PROGRAM MAIN
VAR
fbProfiler: Profiler;
stProfilerResult:PROFILERSTRUCT;
nAnsOfFactorial:ULINT;
END_VAR

fbProfiler(start:=TRUE,reset:=FALSE);
	Factorial(nAnsOfFactorial);	
fbProfiler(start:=FALSE);
stProfilerResult:= fbProfiler.DATA;

END_PROGRAM

(* stored: Version 1.1.0.1, ProductVersion 3.1.4024.12
   POU MAIN: Id {330de865-9760-40d1-98ab-80519ef6e06f}, SpecialFunc None *)
